{attribute addProperty BoxType "AT2041-0250-0019"}
{attribute addProperty Id "A_0103_AT2042_5250_0018_AT2042_5250AT2042_3DCFC8D064080"}
{attribute addProperty CRC "1600510001"}
{attribute addProperty SizeInBites "640"}
{attribute addProperty SizeInBytes "80"}
TYPE A_0041_AT2041_0250_0019_5F65D831 EXTENDS AT2041_9506A482 :
STRUCT
	{attribute addProperty Name "A_0103_AT2042_5250_0018_AT2042_5250"}
	A_0103_AT2042_5250_0018_AT2042_5250 : AT2042_3DCFC8D0;
END_STRUCT
END_TYPE

(* stored: Version 1.2.0.0, ProductVersion 3.1.4024.9
   DUT A_0041_AT2041_0250_0019_5F65D831: Id {6c20ac29-861d-4523-8432-d697e82d6eeb} *)
